//==================================================================================================
//								RJM Maszyny sp. z o.o.
//									13.05.2022
//
//	Obsługa czujnika
//	v1.0	|| TC v 3.1.4024.22		|| - pierwsza wersja
//==================================================================================================
FUNCTION_BLOCK FB_Czujnik_NC IMPLEMENTS I_Czujnik
VAR
	Wejscie							AT %I*	: BOOL;
END_VAR

//==================================================================================================
//								RJM Maszyny sp. z o.o.
//									13.05.2022
//
//	Sprawdzenie czy aktywny
//	v1.0	|| TC v 3.1.4024.22		|| - pierwsza wersja
//==================================================================================================
PROPERTY CzyAktywny : BOOL
GET
CzyAktywny									:= NOT Wejscie;
END_GET
END_PROPERTY

END_FUNCTION_BLOCK

(* stored: Version 1.1.0.1, ProductVersion 3.1.4024.11
   POU FB_Czujnik_NC: Id {cf71bb48-c781-4807-8d04-665179bd48af}, SpecialFunc None
   Property CzyAktywny: Id {d2eae55c-1b03-40b5-949c-64ef2ee19fda}
   Get Get: Id {13e30e11-5125-485e-ade0-0eaac6243855} *)
